# EPICS IOC start-up script: iocsh/sis8300ku.iocsh
#- ###   ESS MTCA IOxOS IFC 14xx iocsh              ###
#- ####################################################
#- >> Mandatory
#- SESS           - SESSION NAME  (MUST BE lowercase)
#- PREF           - PREFIX for the naming
#- UNIT           - UNIT
#- FRUID          - FRUID
#- >> Optional
#- ID             - Default ID, Default : "8300KU"
#- ####################################################

dbLoadRecords("sis8300ku_ess.db", "_PREF=$(PREF), _SESS=$(SESS), _UNIT=$(UNIT), _FRUID=$(FRUID), _ID=$(ID=8300KU)")
#-
